(* CODESYS project PackML_Example.project
   Title: PackML Example
   Version: 1.0.0.0
   Author: 3S - Smart Software Solutions GmbH
   Description: Example project for the PackML State Machine library.
   Company: 3S - Smart Software Solutions GmbH

Project tree, tasks and I/O mapping:
  Device : CODESYS SoftMotion Win V3, 3S - Smart Software Solutions GmbH, order no. 309021, version 3.5.10.0
    application PackMLUnitModeManager
      libraries: Standard, 3.5.18.0 (System); OMAC PackML State Machine, 1.0.0.4 (3S - Smart Software Solutions GmbH); SM3_Robotics, * (CODESYS); SM3_Robotics_Visu, * (CODESYS); SM3_Transformation, * (CODESYS); SM3_Basic, * (CODESYS); Tc3_PackML_V2, 3.3.15.0 (Beckhoff Automation GmbH)
      task MainTask (cyclic, interval t#20ms, priority 1) calls PLC_PRG
      task VISU_TASK (cyclic, interval 100 ms, priority 31) calls VisuElems.Visu_Prg
      program PLC_PRG [ST]: SimulateActingStateComplete
      visualisation Visualization
      global variables GVL
      image pool ImagePool
      PackML/
        global variables G_PML
        PackTags/
          data type PMLs
          Common/
            data type ST_EquipmentInterlock
            data type ST_Descriptor
            data type ST_Alarm
            data type ST_Count
            data type ST_Ingredient
            data type ST_Interface
            data type ST_Product
          data type ST_PMLa
          data type ST_PMLc
        State and Mode/
          data type E_PMLCommand
          data type E_PMLStatus
          data type ST_PMLSubUnitInfo
        ITFs/
          interface I_UnitStateWaiting: M_Aborted, M_Complete, M_Idle, M_Held, M_Stopped, M_Suspended, M_Undefined
          interface I_UnitStateActing: M_Aborting, M_Clearing, M_Completing, M_Execute, M_Holding, M_Reseting, M_Starting, M_StateComplete, M_Stopping, M_Suspending, M_Unholding, M_Unsuspending
          interface I_UnitState: M_Aborting, M_Clearing, M_Completing, M_Execute, M_Holding, M_Reseting, M_Starting, M_StateComplete, M_Stopping, M_Suspending, M_Unholding, M_Unsuspending, M_Aborted, M_Complete, M_Held, M_Idle, M_Stopped, M_Suspended, M_Undefined
        Machine State/
          function block PML_UnitModeConfig [FBD]
          function block PMC_UnitModeManager [FBD]
          function block PML_StateMachine [FBD]
    SoftMotion General Axis Pool
      Axis : SM_Drive_Virtual, 3S - Smart Software Solutions GmbH, order no. 1805, version 4.0.0.0
          settings: iMovementType = 0; fSWMaxVelocity = 1e3; fSWMaxAcceleration = 1e5; fSWMaxDeceleration = 1e5
  Device2 : CODESYS SoftMotion Win V3, 3S - Smart Software Solutions GmbH, order no. 309021, version 3.5.10.0
    application PackMLAxisControl
      libraries: OMAC PackML State Machine, 1.0.0.4 (3S - Smart Software Solutions GmbH)
      task Task (cyclic, interval t#20ms, priority 1) calls PLC_PRG
      task VISU_TASK (cyclic, interval 100 ms, priority 31) calls VisuElems.Visu_Prg
      function block AxisControl [ST]
      program PLC_PRG [ST]
      visualisation Visualization
      image pool ImagePool
    SoftMotion General Axis Pool
      Axis : SM_Drive_Virtual, 3S - Smart Software Solutions GmbH, order no. 1805, version 4.0.0.0
          settings: iMovementType = 0; fSWMaxVelocity = 1e3; fSWMaxAcceleration = 1e5; fSWMaxDeceleration = 1e5
  libraries: VisuSymbols, 4.5.0.0 (System)
  text list GlobalTextList
  5ce3da45-db07-42e7-a21c-a00fff4ed8f6|C:\Users\a.werner\Documents\background.jpg
*)

// Device/PackMLUnitModeManager/PackML/PackTags/PMLs
TYPE PMLs :
STRUCT
	/// 
	///Numeric representation of the active unit mode (required) 
	UnitModeCurrent: DINT; 
	/// 
	///Handshaking bit acknowledging that unit mode change request has been made. 
	UnitModeRequested: BOOL; 
	/// 
	///Signals that unit mode change request has been accepted; switching is actively in process. 
	UnitModeChangeInProcess: BOOL; 
	/// 
	///Numeric representation of the active state (required) 
	StateCurrent: DINT; 
	/// 
	///Handshaking value acknowledging that state change request has been made. 
	StateRequested: DINT; 
	/// 
	///Signals that state change request has been accepted; switching is actively in process. 
	StateChangeInProcess: BOOL; 
	/// 
	///Active machine speed setpoint in units of [primary packages/min] (required) 
	MachSpeed: REAL; 
	/// 
	///Actual machine speed in units of [primary packages/min] (required) 
	CurMachSpeed: REAL; 
	/// 
	///Bitwise indication that materials are ready for processing. 
	MaterialInterlock: ARRAY[0..31] OF BOOL; 
	/// 
	///Signals that the machine is either blocked or starved (required) 
	EquipmentInterlock: ST_EquipmentInterlock; 
	/// 
	///Use to coordinate activities between peers (i.e. upstream or downstream unit machines.) 
	RemoteInterface: ARRAY [1..MaxStatusRemoteInterfaces] OF ST_Interface; 
	/// 
	///Current values or parameters associated to the end user supervisory interface. 
	Parameter: ARRAY [1..MaxStatusParameters] OF ST_Descriptor; 
	/// 
	///Current recipe or process data associated to the various products run on the unit machine. 
	Product: ARRAY [1..MaxStatusProducts] OF ST_Product;	
END_STRUCT
END_TYPE

// Device/PackMLUnitModeManager/PackML/PackTags/Common/ST_EquipmentInterlock
TYPE ST_EquipmentInterlock :
STRUCT
	/// 
	///Machine stoppage due to downstream fault 
	Blocked: BOOL; 
	/// 
	///Machine stoppage due to upstream or supply fault 
	Starved: BOOL;
END_STRUCT
END_TYPE

// Device/PackMLUnitModeManager/PackML/PackTags/Common/ST_Descriptor
TYPE ST_Descriptor :
STRUCT
	 /// 
	 ///Parameter identification number 
	 ID: DINT; 
	 /// 
	 ///Parameter description 
	 Name: STRING; 
	 /// 
	 ///Parameter units of measure 
	 Unit: STRING; 
	 /// 
	 ///Numeric value of parameter 
	 Value: REAL;
END_STRUCT
END_TYPE

// Device/PackMLUnitModeManager/PackML/PackTags/Common/ST_Alarm
TYPE ST_Alarm: 
STRUCT 
	 /// 
	 ///Alarm or warning current status 
	 Trigger: BOOL; 
	 /// 
	 ///Alarm or warning identification number 
	 ID: DINT; 
	 /// 
	 ///Context specific value associated to given alarm or warning 
	 Value: DINT; 
	 /// 
	 ///Alarm or warning description 
	 Message: STRING; 
	 /// 
	 ///Identification number associated to alarm type or severity 
	 Category: DINT; 
	 /// 
	 ///Time stamp of alarm or warning occurrence. Format year:month:day:hour:min:sec:µsec 
	 DateTime: ARRAY[0..6] OF DINT; 
	 /// 
	 ///Time stamp of alarm or warning acknowledgment. Format year:month:day:hour:min:sec:µsec 
	 AckDateTime: ARRAY[0..6] OF DINT; 
END_STRUCT 
END_TYPE

// Device/PackMLUnitModeManager/PackML/PackTags/Common/ST_Count
TYPE ST_Count :
STRUCT
	 /// 
	 ///Product identification number 
	 ID: DINT; 
	 /// 
	 ///Product description 
	 Name: STRING; 
	 /// 
	 ///Product unit of measure 
	 Unit: STRING; 
	 /// 
	 ///Count since last operator reset 
	 Count: DINT; 
	 /// 
	 ///Count since last accumulative counter reset 
	 AccCount: DINT;
END_STRUCT
END_TYPE

// Device/PackMLUnitModeManager/PackML/PackTags/Common/ST_Ingredient
TYPE ST_Ingredient: 
STRUCT 
	 /// 
	 ///Ingredient identification number 
	 IngredientID: DINT; 
	 /// 
	 ///Parameters associated to given ingredient 
	 Parameter: ARRAY[1..G_PML.MaxIngredientParameters] OF ST_Descriptor; 
END_STRUCT 
END_TYPE

// Device/PackMLUnitModeManager/PackML/PackTags/Common/ST_Interface
TYPE ST_Interface :
STRUCT
	 /// 
	 ///Identification number of upstream or downstream unit machine 
	 Number: DINT; 
	 /// 
	 ///Control command for upstream or downstream machine 
	 ControlCmdNumber: DINT; 
	 /// 
	 ///Control command value associated with ControlCmdNumber 
	 CmdValue: DINT; 
	 /// 
	 ///Parameter data required for peer-to-peer coordination 
	 Parameter: ARRAY[1..G_PML.MaxInterfaceParameters] OF ST_Descriptor;
END_STRUCT
END_TYPE

// Device/PackMLUnitModeManager/PackML/PackTags/Common/ST_Product
TYPE ST_Product :
STRUCT
	 /// 
	 ///Product identification number 
	 ProductID: DINT; 
	 /// 
	 ///Parameters required for processing given product 
	 ProcessVariables: ARRAY[1..G_PML.MaxProductProcessVariables] OF ST_Descriptor; 
	 /// 
	 ///Ingredients required for processing given product 
	 Ingredients: ARRAY[1..G_PML.MaxIngredients] OF ST_Ingredient;	
END_STRUCT
END_TYPE

// Device/PackMLUnitModeManager/PackML/PackTags/ST_PMLa
TYPE ST_PMLa :
STRUCT
	/// 
	///Parameters associated to the local interface (e.g. HMI) 
	Parameter: ARRAY [1..G_PML.MaxAdminParameters] OF ST_Descriptor; 
	/// 
	///Listing of all currently active alarms 
	Alarm: ARRAY [1..G_PML.MaxAlarms] OF ST_Alarm; 
	/// 
	///Extent of the Alarm array 
	AlarmExtent: DINT	:= G_PML.MaxAlarms; 
	/// 
	///Chronological alarm history, with most recent given as AlarmHistory[0] 
	AlarmHistory: ARRAY [1..G_PML.MaxHistoryAlarms] OF ST_Alarm; 
	/// 
	///Extent of AlarmHistory array 
	AlarmHistoryExtent: DINT	:= G_PML.MaxHistoryAlarms; 
	/// 
	///Alarm associated to the primary cause of machine stoppage ('first fault') (required) 
	StopReason: ARRAY [1..G_PML.MaxStopReasons] OF ST_Alarm; 
	/// 
	///Extent of StopReason array 
	StopReasonExtent: DINT	:= G_PML.MaxStopReasons; 
	/// 
	///Listing of all currently active warnings 
	Warning: ARRAY [1..G_PML.MaxWarnings] OF ST_Alarm; 
	/// 
	///Extent of warning array 
	WarningExtent: DINT	:= G_PML.MaxWarnings; 
	/// 
	///Elapsed time in seconds of current mode. 
	ModeCurrentTime: ARRAY [0..G_PML.MaxUnitMode] OF DINT;
	/// 
	///Cumulative time in seconds in each defined mode. 
	ModeCumulativeTime: ARRAY [0..G_PML.MaxUnitMode] OF DINT; 
	/// 
	///Elapsed time in seconds of current [mode, state] pair. 
	StateCurrentTime: ARRAY [0..G_PML.MaxUnitMode, 0..G_PML.MaxMachineState] OF DINT; 
	/// 
	///Cumulative time in seconds in each defined [mode, state] pair. 
	StateCumulativeTime: ARRAY [0..G_PML.MaxUnitMode, 0..G_PML.MaxMachineState] OF DINT; 
	/// 
	///Count of raw materials used or consumed during production 
	ProdConsumedCount: ARRAY [1..G_PML.MaxConsumedCounts] OF ST_Count; 
	/// 
	///Count of total products (i.e. good + defective) made during production (required) 
	ProdProcessedCount: ARRAY [1..G_PML.MaxProductCounts] OF ST_Count; 
	/// 
 	///Count of defective products made during production. (required) 
	ProdDefectiveCount: ARRAY [1..G_PML.MaxProductCounts] OF ST_Count; 
	/// 
	///Accumulative time since last reset of timer arrays. 
	AccTimeSinceReset: DINT; 	
	/// 
	///Maximum design speed of the machine within given environment. 
	MachDesignSpeed: REAL; 	
	/// 
	///Bitwise indication of inactive states in current mode. 
	StatesDisabled: DINT; 		
	/// 
	///Current date and time of local processing unit (PLC, PC, PAC, microcontroller, etc.) 
	PLCDateTime: ARRAY[0..6] OF DINT;
END_STRUCT
END_TYPE

// Device/PackMLUnitModeManager/PackML/PackTags/ST_PMLc
TYPE ST_PMLc :
STRUCT
	/// 
	///Numeric representation of the commanded unit mode (required) 
	UnitMode: DINT; 
	/// 
	///Signals request that the current value of Command.UnitMode be activated (required) 
	UnitModeChangeRequest: BOOL; 
	/// 
	///Machine speed setpoint in units of [primary packages/min] (required) 
	MachSpeed: REAL; 
	/// 
	///Bitwise indication that materials are ready for processing. 
	MaterialInterlock: ARRAY[1..32] OF BOOL; 
	/// 
	///Numerical representation of the state commands (1=Reset, 2=Start, etc.) (required) 
	CntrlCmd: DINT; 
	/// 
	///Signals request that the current value of Command.CntrlCmd be activated (required) 
	CmdChangeRequest: BOOL; 
	///
	///Use to coordinate activities between peers (i.e. upstream or downstream unit machines.) 
	RemoteInterface: ARRAY [1..G_PML.MaxCommandRemoteInterfaces] OF ST_Interface; 
	/// 
	///Values or parameters associated to the end user supervisory interface. 
	Parameter: ARRAY [1..G_PML.MaxCommandParameters] OF ST_Descriptor; 
	/// 
	///Recipe or process data associated to the various products run on the unit machine. 
	Product: ARRAY [1..G_PML.MaxCommandProducts] OF ST_Product;
	
END_STRUCT
END_TYPE

// Device/PackMLUnitModeManager/PackML/State and Mode/E_PMLCommand
{attribute 'qualified_only'}
{attribute 'strict'}
TYPE E_PMLCommand :
(
	ePMLCommand_Undefined		:=	0,	
	ePMLCommand_Reset			:=	1,	
	ePMLCommand_Start			:=	2,	
	ePMLCommand_Stop			:=	3,	
	ePMLCommand_Hold			:=	4,	
	ePMLCommand_Unhold			:=	5,	
	ePMLCommand_Suspend			:=	6,	
	ePMLCommand_Unsuspend		:=	7,	
	ePMLCommand_Abort			:=	8,	
	ePMLCommand_Clear			:=	9,	
	//	extension TO OMAC TR88.00.02
	ePMLCommand_Complete		:=	10
);
END_TYPE

// Device/PackMLUnitModeManager/PackML/State and Mode/E_PMLStatus
{attribute 'qualified_only'}
{attribute 'strict'}
TYPE E_PMLStatus :
(
	//states according TO PackTags v3.0
	ePMLState_Undefined		:=			0,	
	ePMLState_Clearing		:=			1,	
	ePMLState_Stopped		:=			2,	
	ePMLState_Starting		:=			3,	
	ePMLState_Idle			:=			4,	
	ePMLState_Suspended		:=			5,	
	ePMLState_Execute		:=			6,	
	ePMLState_Stopping		:=			7,	
	ePMLState_Aborting		:=			8,	
	ePMLState_Aborted		:=			9,	
	ePMLState_Holding		:=			10,	
	ePMLState_Held			:=			11,	
	ePMLState_Unholding		:=			12,	
	ePMLState_Suspending	:=			13,	
	ePMLState_Unsuspending	:=			14,	
	ePMLState_Resetting		:=			15,	
	ePMLState_Completing	:=			16,	
	ePMLState_Complete		:=			17
);
END_TYPE

// Device/PackMLUnitModeManager/PackML/State and Mode/ST_PMLSubUnitInfo
TYPE ST_PMLSubUnitInfo :
STRUCT
	Active	: BOOL;				
	eState	: E_PMLState	:=	ePMLState_Aborted;	
END_STRUCT
END_TYPE

// Device/PackMLUnitModeManager/GVL
VAR_GLOBAL CONSTANT
	gc_sPRODUCTION : STRING := 'Production';
	gc_sSEMIAUTO : STRING := 'Semi Auto';
	gc_sSETUP : STRING := 'Setup';
END_VAR

// Device/PackMLUnitModeManager/PackML/G_PML
{attribute 'qualified_only'}
VAR_GLOBAL CONSTANT
	MaxInterfaceParameters		: INT	:=5	;//PMLc/PMLs
	MaxProductProcessVariables	: INT	:=10;
	MaxIngredients				: INT	:=10;
	MaxIngredientParameters		: INT	:=10;
	MaxCommandRemoteInterfaces	: INT	:=2;	//PMLc
	MaxCommandParameters		: INT	:=10;	
	MaxCommandProducts			: INT	:=5;
	MaxStatusRemoteInterfaces	: INT	:=2;	//PMLs
	MaxStatusParameters			: INT	:=10;	
	MaxStatusProducts			: INT	:=5;	
	MaxAdminParameters			: INT	:=10;	//PMLa
	MaxAlarms					: INT	:=10;	
	MaxHistoryAlarms			: INT	:=10;	
	MaxStopReasons				: INT	:=10;	
	MaxWarnings					: INT	:=10;	
	MaxConsumedCounts			: INT	:=10;	
	MaxProductCounts			: INT	:=10;
	
	MaxUnitMode					:INT	:=31;
	MaxMachineState				:INT	:=17;
	stPMLUnitModeConfiguration	:ARRAY [0..MaxUnitMode] OF ST_PMLUnitModeConfiguration	:=	[STRUCT(bActive := TRUE, sName := 'Invalid', aStateDisabled := [18(FALSE)], aModeChangeValid := [18(TRUE)]), STRUCT(bActive := TRUE, sName := 'Production', aStateDisabled := [18(FALSE)], aModeChangeValid := [TRUE, FALSE, TRUE, FALSE, TRUE, FALSE, FALSE, FALSE, FALSE, TRUE, FALSE, TRUE, FALSE, FALSE, FALSE, FALSE, FALSE, FALSE]), STRUCT(bActive := TRUE, sName := 'Maintenance', aStateDisabled := [FALSE, FALSE, FALSE, FALSE, FALSE, TRUE, FALSE, FALSE, FALSE, FALSE, FALSE, FALSE, FALSE, TRUE, TRUE, FALSE, TRUE, TRUE], aModeChangeValid := [TRUE, FALSE, TRUE, FALSE, TRUE, FALSE, FALSE, FALSE, FALSE, TRUE, FALSE, TRUE, FALSE, FALSE, FALSE, FALSE, FALSE, FALSE]), STRUCT(bActive := TRUE, sName := 'Manual', aStateDisabled := [FALSE, FALSE, FALSE, FALSE, FALSE, TRUE, FALSE, FALSE, FALSE, FALSE, TRUE, TRUE, TRUE, TRUE, TRUE, FALSE, TRUE, TRUE], aModeChangeValid := [TRUE, FALSE, TRUE, FALSE, TRUE, FALSE, FALSE, FALSE, FALSE, TRUE, FALSE, FALSE, FALSE, FALSE, FALSE, FALSE, FALSE, FALSE])];	

	
END_VAR

// Device/PackMLUnitModeManager/PLC_PRG
// Example project for the PackML State Machine with three unit modes.
PROGRAM PLC_PRG
VAR
	productionUnitMode	: PACK_ML.UnitMode; // Example unit mode for prodction
	semiAutoUnitMode	: PACK_ML.UnitMode; // Example unit mode for semi auto production
	setupUnitMode		: PACK_ML.UnitMode; // Example unit mode for setup
	unitModeManager		: PACK_ML.UnitModeManager; // Unit mode manager to switch between unitmodes
	currentUnitMode		: PACK_ML.IUnitMode;
	xInit				: BOOL := FALSE; // Flag for initialization
	
	// Visu Commands	
	xAbort				: BOOL;
	xActingStateComplete: BOOL;
	xClear				: BOOL;
	xHold				: BOOL;
	xReset				: BOOL;
	xStart				: BOOL;
	xStop				: BOOL;
	xSuspend			: BOOL;
	xUnHold				: BOOL;
	xUnSuspend			: BOOL;
	
	// Helper
	xSimulate			: BOOL;
	xChangeState		: BOOL := FALSE;	
	timer1				: TON;	
	iSelectedUnitMode	: INT := 0;
	iLastSelectedUnitMode: INT := 0;
	xUserModeChanged	: BOOL;
END_VAR

IF NOT xInit THEN
	productionUnitMode(		sName := gc_sPRODUCTION, 
							dwSupportedStates := PACK_ML.State.All, 
							dwAllowsLeavingFromStates := PACK_ML.State.Stopped OR PACK_ML.State.Aborted OR PACK_ML.State.Idle, 
							dwAllowsEnteringIntoStates := PACK_ML.State.Stopped OR PACK_ML.State.Aborted OR PACK_ML.State.Idle, 
							eInitialState := PACK_ML.State.Idle,
							xActive := TRUE);
	semiAutoUnitMode(		sName := gc_sSEMIAUTO, 
							dwSupportedStates := PACK_ML.State.All - PACK_ML.State.Completing - PACK_ML.State.Complete - PACK_ML.State.Holding - PACK_ML.State.Held - PACK_ML.State.UnHolding,
							dwAllowsLeavingFromStates := PACK_ML.State.Stopped OR PACK_ML.State.Aborted OR PACK_ML.State.Idle, 
							dwAllowsEnteringIntoStates := PACK_ML.State.Stopped OR PACK_ML.State.Aborted OR PACK_ML.State.Idle,   
							eInitialState := PACK_ML.State.Idle, 
							xActive := FALSE);
	setupUnitMode(			sName := gc_sSETUP, 
							dwSupportedStates := PACK_ML.State.All - PACK_ML.State.Completing - PACK_ML.State.Complete - PACK_ML.State.Holding - PACK_ML.State.Held - PACK_ML.State.UnHolding - PACK_ML.State.UnSuspending - PACK_ML.State.Suspended - PACK_ML.State.Suspending,
							dwAllowsLeavingFromStates := PACK_ML.State.Stopped OR PACK_ML.State.Aborted OR PACK_ML.State.Idle,   
							dwAllowsEnteringIntoStates := PACK_ML.State.Stopped OR PACK_ML.State.Aborted OR PACK_ML.State.Idle, 
							eInitialState := PACK_ML.State.Idle, 
							xActive := FALSE);

	// Register the unit modes 
	unitModeManager.Register(productionUnitMode);
	unitModeManager.Register(semiAutoUnitMode);
	unitModeManager.Register(setupUnitMode);
	xInit := TRUE;
END_IF

IF unitModeManager.ActiveUnitMode <> 0 THEN	
	currentUnitMode := unitModeManager.ActiveUnitMode;
	
	// Visu commands
	IF xAbort THEN
		unitModeManager.ActiveUnitMode.Abort();
	END_IF
	IF xClear THEN
		unitModeManager.ActiveUnitMode.Clear();
	END_IF
	IF xHold THEN
		unitModeManager.ActiveUnitMode.Hold();
	END_IF
	IF xReset THEN
		unitModeManager.ActiveUnitMode.Reset();
	END_IF
	IF xStart THEN
		unitModeManager.ActiveUnitMode.Start();
	END_IF
	IF xStop THEN
		unitModeManager.ActiveUnitMode.Stop();
	END_IF
	IF xSuspend THEN
		unitModeManager.ActiveUnitMode.Suspend();
	END_IF
	IF xUnHold THEN
		unitModeManager.ActiveUnitMode.UnHold();
	END_IF
	IF xUnSuspend THEN
		unitModeManager.ActiveUnitMode.UnSuspend();
	END_IF
	IF xActingStateComplete AND NOT xSimulate THEN
		unitModeManager.ActiveUnitMode.ActingStateCompleted();
	END_IF
	
	// Simulate action complete
	SimulateActingStateComplete();	 
END_IF

// Change the current unit mode
IF iSelectedUnitMode <> iLastSelectedUnitMode THEN
	IF iSelectedUnitMode = 0 THEN
		xUserModeChanged := unitModeManager.SwitchUnitMode(gc_sPRODUCTION);
	ELSIF iSelectedUnitMode = 1 THEN
		xUserModeChanged := unitModeManager.SwitchUnitMode(gc_sSEMIAUTO);
	ELSE
 		xUserModeChanged := unitModeManager.SwitchUnitMode(gc_sSETUP);
	END_IF
	IF xUserModeChanged THEN
		iLastSelectedUnitMode := iSelectedUnitMode;
	ELSE
		iSelectedUnitMode := iLastSelectedUnitMode;
	END_IF
END_IF

METHOD SimulateActingStateComplete
VAR_INPUT
END_VAR
VAR
	nextSupportedState	: UDINT;	
END_VAR
nextSupportedState := unitModeManager.ActiveUnitMode.NextState(unitModeManager.ActiveUnitMode.CurrentState);	
IF nextSupportedState = PACK_ML.State.Execute OR nextSupportedState = PACK_ML.State.Completing OR nextSupportedState = PACK_ML.State.Complete OR nextSupportedState = PACK_ML.State.Held OR nextSupportedState = PACK_ML.State.Aborted OR nextSupportedState = PACK_ML.State.Stopped OR nextSupportedState = PACK_ML.State.Idle OR nextSupportedState = PACK_ML.State.Suspended THEN	
	timer1(IN := TRUE, PT := T#2S, Q => xChangeState);
	xSimulate := TRUE;
END_IF   
IF xChangeState THEN
	unitModeManager.ActiveUnitMode.ActingStateCompleted();
	timer1(IN := FALSE);
	xSimulate := FALSE;
	xChangeState := FALSE;
END_IF
END_METHOD

END_PROGRAM

// Device2/PackMLAxisControl/PLC_PRG
PROGRAM PLC_PRG
VAR
	xInit				: BOOL := FALSE; // Flag for initialization

	ac: AxisControl;
	
	// Visu Commands	
	xAbort				: BOOL;
	xActingStateComplete: BOOL;
	xClear				: BOOL;
	xHold				: BOOL;
	xReset				: BOOL;
	xStart				: BOOL;
	xStop				: BOOL;
	xSuspend			: BOOL;
	xUnHold				: BOOL;
	xUnSuspend			: BOOL;
	
	
END_VAR

ac(Axis:=Axis);

// Visu commands
IF xAbort THEN
	ac.ItfUnitMode.Abort();
END_IF
IF xClear THEN
	ac.ItfUnitMode.Clear();
END_IF
IF xHold THEN
	ac.ItfUnitMode.Hold();
END_IF
IF xReset THEN
	ac.ItfUnitMode.Reset();
END_IF
IF xStart THEN
	ac.ItfUnitMode.Start();
END_IF
IF xStop THEN
	ac.ItfUnitMode.Stop();
END_IF
IF xSuspend THEN
	ac.ItfUnitMode.Suspend();
END_IF
IF xUnHold THEN
	ac.ItfUnitMode.UnHold();
END_IF
IF xUnSuspend THEN
	ac.ItfUnitMode.UnSuspend();
END_IF
IF xActingStateComplete AND ac.ItfUnitMode.CurrentState = PACK_ML.State.Execute THEN
	ac.ItfUnitMode.ActingStateCompleted();
END_IF

END_PROGRAM

// Device2/PackMLAxisControl/AxisControl
FUNCTION_BLOCK AxisControl
// This FB represents an axis, which is controlled according to its active unit mode
VAR_IN_OUT
	Axis: AXIS_REF_SM3;
END_VAR
VAR_OUTPUT
	ItfUnitMode	: PACK_ML.IUnitMode; // UnitMode of the axis
END_VAR
VAR
	UM	: PACK_ML.UnitMode; 

	xInit				: BOOL := FALSE; // Flag for initialization

	//motion FBs
	p: MC_Power;
	rs: MC_ReadStatus;
	res: MC_Reset;
	moverel: MC_MoveRelative;
	halt: MC_Halt;
	moveabs: MC_MoveAbsolute;
	h: MC_Home;
END_VAR

IF NOT xInit THEN	
	UM				(		sName := 'Normal Operation', 
							dwSupportedStates := PACK_ML.State.All - PACK_ML.State.Suspending - PACK_ML.State.Suspended - PACK_ML.State.UnSuspending, 
							dwAllowsLeavingFromStates := PACK_ML.State.Stopped OR PACK_ML.State.Aborted OR PACK_ML.State.Idle, 
							dwAllowsEnteringIntoStates := PACK_ML.State.Stopped OR PACK_ML.State.Aborted OR PACK_ML.State.Idle, 
							eInitialState := PACK_ML.State.Aborted,
							xActive := TRUE);
	ItfUnitMode := UM; 
	xInit := TRUE;
END_IF

CASE UM.CurrentState OF
PACK_ML.State.Stopped,
PACK_ML.State.Aborted,
PACK_ML.State.Idle,
PACK_ML.State.Held,
PACK_ML.State.Complete :
	// in this waiting states we reset the Execute input of the moving FBs
	res.Execute := FALSE;
	moverel.Execute := FALSE;
	halt.Execute := FALSE;
	moveabs.Execute := FALSE;
	h.Execute := FALSE;
PACK_ML.State.Resetting :
	IF rs.Errorstop THEN	//first reset errors when necessary
		h.Execute := FALSE;
		IF res.Error THEN
			res.Execute := FALSE;
		ELSE	
			res.Execute := TRUE;
		END_IF
	ELSE
		p.bDriveStart := TRUE;	//release quickstop
		IF p.Status THEN
			h.Execute := TRUE;	//do homing
			IF h.Done THEN	
				h.Execute := FALSE;
				UM.ActingStateCompleted();
			END_IF
		END_IF
	END_IF
PACK_ML.State.Starting :
	moverel.Execute:=FALSE;
	UM.ActingStateCompleted();
PACK_ML.State.Execute :
	moverel.Execute:=TRUE;
	IF moverel.Done THEN
		moverel.Execute:=FALSE;
 	END_IF
PACK_ML.State.Holding :
	moverel.Execute:=FALSE;
	halt.Execute:=TRUE;
	IF halt.Done THEN
		halt.Execute := FALSE;
		UM.ActingStateCompleted();
	END_IF
PACK_ML.State.UnHolding :
	halt.Execute:=FALSE;
	moveabs.Execute := TRUE;
	IF moveabs.Done THEN
		moveabs.Execute := FALSE;
		UM.ActingStateCompleted();
	END_IF
PACK_ML.State.Completing :
	IF moverel.Done THEN
		UM.ActingStateCompleted();
	END_IF
PACK_ML.State.Aborting :
	p.bDriveStart := FALSE;
	p.bRegulatorOn := FALSE;
	UM.ActingStateCompleted();
PACK_ML.State.Stopping,
PACK_ML.State.Clearing :	
	p.bRegulatorOn:=TRUE; 
	p.bDriveStart:=FALSE; 
	IF p.bRegulatorRealState AND NOT p.bDriveStartRealState THEN
		UM.ActingStateCompleted();
	END_IF
END_CASE

p(
	Axis:=Axis , 
	Enable:=TRUE , 
	Status=> , 
	bRegulatorRealState=> , 
	bDriveStartRealState=> , 
	Busy=> , 
	Error=> , 
	ErrorID=> );

rs(
	Axis:=Axis , 
	Enable:=TRUE , 
	Valid=> , 
	Busy=> , 
	Error=> , 
	ErrorID=> , 
	Disabled=> , 
	Errorstop=> , 
	Stopping=> , 
	StandStill=> , 
	DiscreteMotion=> , 
	ContinuousMotion=> , 
	SynchronizedMotion=> , 
	Homing=> , 
	ConstantVelocity=> , 
	Accelerating=> , 
	Decelerating=> , 
	FBErrorOccured=> );
	
res(
	Axis:=Axis , 
	Execute:= , 
	Done=> , 
	Busy=> , 
	Error=> , 
	ErrorID=> );
	
moverel(
	Axis:=Axis , 
	Distance:=360 , 
	Velocity:=360 , 
	Acceleration:=360 , 
	Deceleration:=360, 
	Jerk:= , 
	Done=> , 
	Busy=> , 
	CommandAborted=> , 
	Error=> , 
	ErrorID=> );
	
moveabs(
	Axis:=Axis , 
	Execute:= , 
	Position:=0 , 
	Velocity:=360 , 
	Acceleration:=360 , 
	Deceleration:=360 , 
	Jerk:= , 
	Direction:=positive , 
	Done=> , 
	Busy=> , 
	CommandAborted=> , 
	Error=> , 
	ErrorID=> );
	
halt(
	Axis:=axis , 
	Execute:= , 
	Deceleration:=1000 , 
	Jerk:= , 
	Done=> , 
	Busy=> , 
	CommandAborted=> , 
	Error=> , 
	ErrorID=> );
	
h(
	Axis:=Axis , 
	Execute:= , 
	Position:= , 
	Done=> , 
	Busy=> , 
	CommandAborted=> , 
	Error=> , 
	ErrorID=> );

END_FUNCTION_BLOCK

// Device/PackMLUnitModeManager/PackML/ITFs/I_UnitStateWaiting
INTERFACE I_UnitStateWaiting

METHOD M_Aborted
VAR_INPUT
END_VAR
END_METHOD

METHOD M_Complete
VAR_INPUT
END_VAR
END_METHOD

METHOD M_Idle
VAR_INPUT
END_VAR
END_METHOD

METHOD M_Held
VAR_INPUT
END_VAR
END_METHOD

METHOD M_Stopped
VAR_INPUT
END_VAR
END_METHOD

METHOD M_Suspended
VAR_INPUT
END_VAR
END_METHOD

METHOD M_Undefined
VAR_INPUT
END_VAR
END_METHOD

END_INTERFACE

// Device/PackMLUnitModeManager/PackML/ITFs/I_UnitStateActing
INTERFACE I_UnitStateActing

METHOD M_Aborting
VAR_INPUT
END_VAR
END_METHOD

METHOD M_Clearing
VAR_INPUT
END_VAR
END_METHOD

METHOD M_Completing
VAR_INPUT
END_VAR
END_METHOD

METHOD M_Execute
VAR_INPUT
END_VAR
END_METHOD

METHOD M_Holding
VAR_INPUT
END_VAR
END_METHOD

METHOD M_Reseting
VAR_INPUT
END_VAR
END_METHOD

METHOD M_Starting
VAR_INPUT
END_VAR
END_METHOD

METHOD M_StateComplete
VAR_INPUT
END_VAR
END_METHOD

METHOD M_Stopping
VAR_INPUT
END_VAR
END_METHOD

METHOD M_Suspending
VAR_INPUT
END_VAR
END_METHOD

METHOD M_Unholding
VAR_INPUT
END_VAR
END_METHOD

METHOD M_Unsuspending
VAR_INPUT
END_VAR
END_METHOD

END_INTERFACE

// Device/PackMLUnitModeManager/PackML/ITFs/I_UnitState
INTERFACE I_UnitState EXTENDS I_UnitStateWaiting,I_UnitStateActing

METHOD M_Aborting
VAR_INPUT
END_VAR
END_METHOD

METHOD M_Clearing
VAR_INPUT
END_VAR
END_METHOD

METHOD M_Completing
VAR_INPUT
END_VAR
END_METHOD

METHOD M_Execute
VAR_INPUT
END_VAR
END_METHOD

METHOD M_Holding
VAR_INPUT
END_VAR
END_METHOD

METHOD M_Reseting
VAR_INPUT
END_VAR
END_METHOD

METHOD M_Starting
VAR_INPUT
END_VAR
END_METHOD

METHOD M_StateComplete
VAR_INPUT
END_VAR
END_METHOD

METHOD M_Stopping
VAR_INPUT
END_VAR
END_METHOD

METHOD M_Suspending
VAR_INPUT
END_VAR
END_METHOD

METHOD M_Unholding
VAR_INPUT
END_VAR
END_METHOD

METHOD M_Unsuspending
VAR_INPUT
END_VAR
END_METHOD

METHOD M_Aborted
VAR_INPUT
END_VAR
END_METHOD

METHOD M_Complete
VAR_INPUT
END_VAR
END_METHOD

METHOD M_Held
VAR_INPUT
END_VAR
END_METHOD

METHOD M_Idle
VAR_INPUT
END_VAR
END_METHOD

METHOD M_Stopped
VAR_INPUT
END_VAR
END_METHOD

METHOD M_Suspended
VAR_INPUT
END_VAR
END_METHOD

METHOD M_Undefined
VAR_INPUT
END_VAR
END_METHOD

END_INTERFACE

// Device/PackMLUnitModeManager/PackML/Machine State/PML_UnitModeConfig
FUNCTION_BLOCK PML_UnitModeConfig
VAR_INPUT
	//
	eMode							: DINT;				
	sName							: STRING;
	//config which state disable				
	bDisableClearing				: BOOL;				
	bDisableStarting				: BOOL;				
	bDisableSuspended				: BOOL;				
	bDisableStopping				: BOOL;				
	bDisableAborting				: BOOL;				
	bDisableHolding					: BOOL;				
	bDisableHeld					: BOOL;				
	bDisableUnholding				: BOOL;				
	bDisableSuspending				: BOOL;				
	bDisableUnsuspending			: BOOL;				
	bDisableResetting				: BOOL;				
	bDisableIdle					: BOOL;				
	bDisableCompleting				: BOOL;				
	bDisableComplete				: BOOL;
	//config unit mode can be changed in which state				
	bEnableUnitModeChangeStopped	: BOOL;				
	bEnableUnitModeChangeIdle		: BOOL;				
	bEnableUnitModeChangeSuspended	: BOOL;				
	bEnableUnitModeChangeExecute	: BOOL;				
	bEnableUnitModeChangeAborted	: BOOL;				
	bEnableUnitModeChangeHeld		: BOOL;				
	bEnableUnitModeChangeComplete	: BOOL;		
END_VAR
VAR_OUTPUT
	bError	: BOOL;				
	nErrorId	: UDINT;	
END_VAR
VAR
END_VAR

// NETWORK 1

END_FUNCTION_BLOCK

// Device/PackMLUnitModeManager/PackML/Machine State/PMC_UnitModeManager
FUNCTION_BLOCK PMC_UnitModeManager
VAR_INPUT
END_VAR
VAR_OUTPUT
END_VAR
VAR
END_VAR

// NETWORK 1

END_FUNCTION_BLOCK

// Device/PackMLUnitModeManager/PackML/Machine State/PML_StateMachine
FUNCTION_BLOCK PML_StateMachine
VAR_INPUT
END_VAR
VAR_OUTPUT
END_VAR
VAR
END_VAR

// NETWORK 1

END_FUNCTION_BLOCK

// Device/PackMLUnitModeManager/Visualization
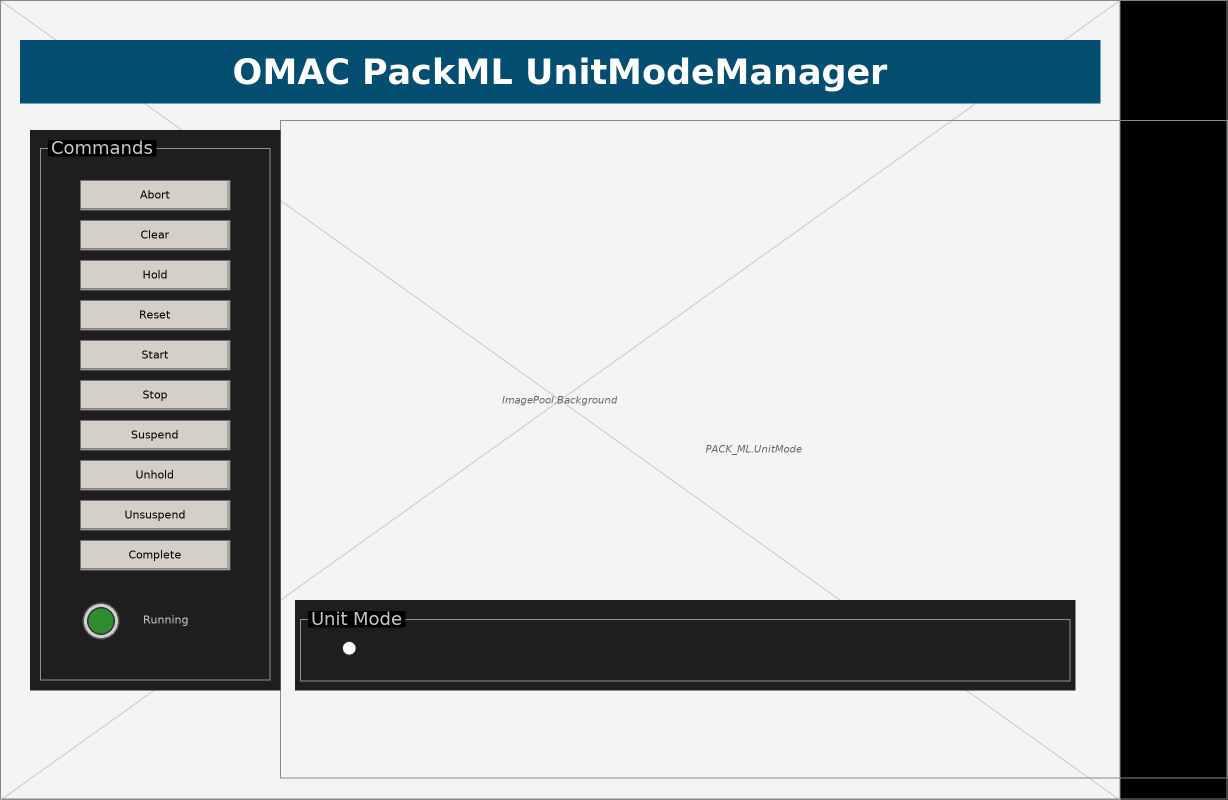
VISUALIZATION Visualization  // 1228x800
    Image (0,0 1120x800), image: ImagePool.Background
    Frame (280,120 948x658)
        shows PACK_ML.UnitMode(um := PLC_PRG.currentUnitMode)
    Rectangle (295,600 780x90)
    Rectangle (30,130 250x560)
    GroupBox (40,140 230x540), "Commands"
        Lamp1 (40,460 42x42), variable: PLC_PRG.xSimulate, style: Lamp-Lamp1-Green
        Label (100,465 57x30), "Running"
        Button (40,40 150x30), "Abort"
            tap PLC_PRG.xAbort
        Button (40,80 150x30), "Clear"
            tap PLC_PRG.xClear
        Button (40,120 150x30), "Hold"
            tap PLC_PRG.xHold
        Button (40,160 150x30), "Reset"
            tap PLC_PRG.xReset
        Button (40,200 150x30), "Start"
            tap PLC_PRG.xStart
        Button (40,240 150x30), "Stop"
            tap PLC_PRG.xStop
        Button (40,280 150x30), "Suspend"
            tap PLC_PRG.xSuspend
        Button (40,320 150x30), "Unhold"
            tap PLC_PRG.xUnHold
        Button (40,360 150x30), "Unsuspend"
            tap PLC_PRG.xUnSuspend
        Button (40,400 150x30), "Complete"
            tap PLC_PRG.xActingStateComplete
    GroupBox (300,611 770x70), "Unit Mode"
        RadioButton (40,20 700x34), variable: PLC_PRG.iSelectedUnitMode
            Areas[0]: Text=Production
            Areas[1]: Text=Semi Auto Production
            Areas[2]: Text=Setup
    Rectangle (20,40 1080x63), "OMAC PackML UnitModeManager"
END_VISUALIZATION

// Device2/PackMLAxisControl/Visualization
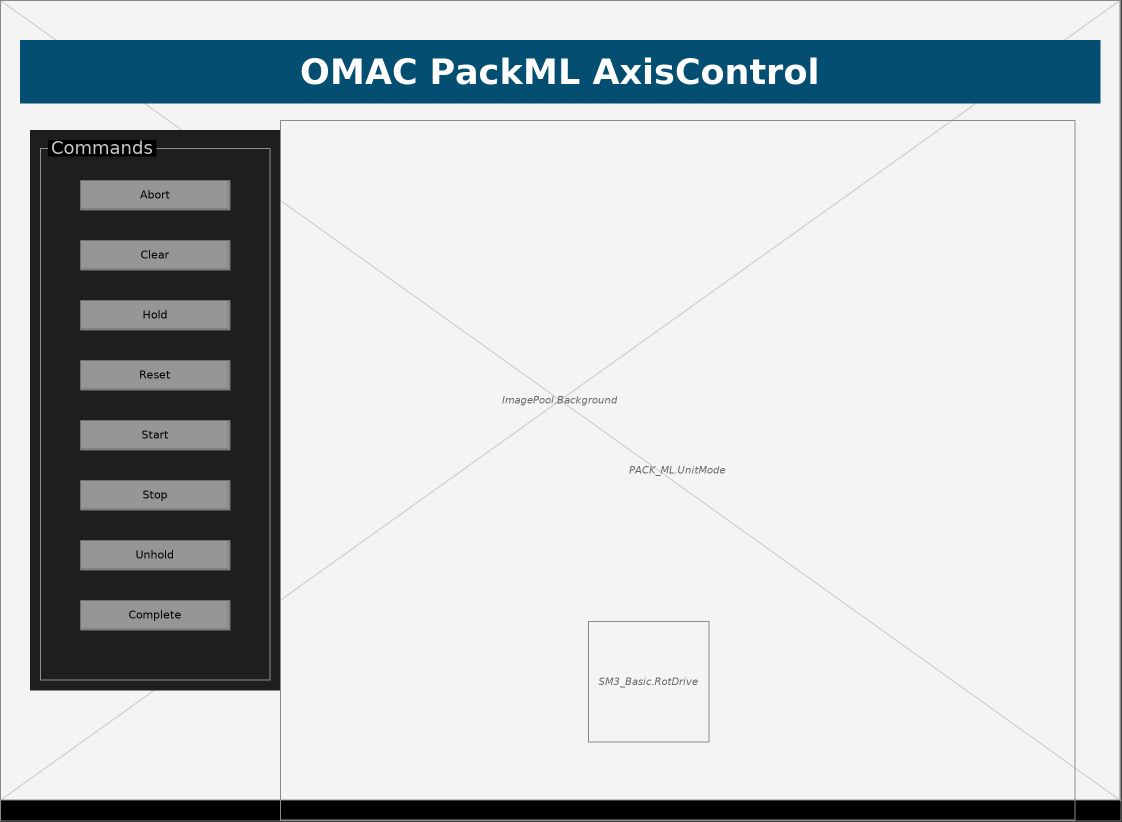
VISUALIZATION Visualization  // 1122x822
    Image (0,0 1120x800), image: ImagePool.Background
    Rectangle (30,130 250x560)
    GroupBox (40,140 230x540), "Commands"
        Button (40,40 150x30), "Abort"
            tap PLC_PRG.xAbort
        Button (40,100 150x30), "Clear"
            tap PLC_PRG.xClear
        Button (40,160 150x30), "Hold"
            tap PLC_PRG.xHold
        Button (40,220 150x30), "Reset"
            tap PLC_PRG.xReset
        Button (40,280 150x30), "Start"
            tap PLC_PRG.xStart
        Button (40,340 150x30), "Stop"
            tap PLC_PRG.xStop
        Button (40,400 150x30), "Unhold"
            tap PLC_PRG.xUnHold
        Button (40,460 150x30), "Complete"
            tap PLC_PRG.xActingStateComplete
    Frame (280,120 795x700)
        shows PACK_ML.UnitMode(um := PLC_PRG.ac.UM)
    Frame (588,621 121x121)
        shows SM3_Basic.RotDrive(m_Input_AXISREF := Axis)
    Rectangle (20,40 1080x63), "OMAC PackML AxisControl"
END_VISUALIZATION
